// Mitsubishi GX Works2 project: EX_2_GROUP10   PLC: FX3G

// global labels: Global1
VAR_GLOBAL
  hopsInput AT D1120 : REAL;  (* input for hops inventory *)
  yeastQuantity AT D1130 : REAL;  (* yeast current quantity *)
  hopsQuantity AT D1150 : REAL;  (* hops current quantity *)
  startCooking AT X001 : BOOL;  (* starting stage 1 - cooking *)
  enoughIngredients AT M4 : BOOL;  (* if there is not quantity problem (enough required ingredients) *)
END_VAR
VAR_GLOBAL CONSTANT
  fermentationPilsnerTime : INT := 40;  (* fermentation time of Pilsner beer *)
  fermentationLagerTime : INT := 30;  (* fermentation time of Lager beer *)
  cookTime : INT := 40;  (* beer cook time last 4 seconds *)
  constant_0 : REAL;  (* constant zero *)
END_VAR
VAR_GLOBAL
  sampleValue AT D8201 : INT;  (* Sample value which symbolize the type of selected beer *)
END_VAR
VAR_GLOBAL CONSTANT
  normaliztionFactor : INT := 400;  (* normaliztion factor for the sampled value of beer kind *)
  maxLager : INT := 6;  (* Minimum sample value for lager beer (Underneath it is necessarily Pilsner beer) *)
  barleyLager : REAL := 12;  (* minimum quantity needed of barley for Lager beer *)
  hopsLager : REAL := 60;  (* minimum quantity needed of hops for Lager beer *)
  yeastPilsner : REAL := 120;  (* minimum quantity needed of yeast for Pilsner beer *)
  barleyPilsner : REAL := 6;  (* minimum quantity needed of barley for Pilsner beer *)
  hopsPilsner : REAL := 53;  (* minimum quantity needed of hops for Pilsner beer *)
END_VAR
VAR_GLOBAL
  barleyInput AT D1110 : REAL;  (* input for barley inventory *)
  yeastInput AT D1100 : REAL;  (* input for yeast inventory *)
  startDay AT X007 : BOOL;  (* start day button *)
  barleyQuantity AT D1140 : REAL;  (* barley current quantity *)
  yeast46Beers AT D1160 : REAL;  (* yeast demand for 6 beers *)
  barley46Beers AT D1170 : REAL;  (* barley demand for 6 beers *)
  cookContainer AT D2010 : REAL;  (* current quantity of raw materials in the cooking container *)
  emergencyButton AT X011 : BOOL;  (* emergency button that stopping the day (production process) *)
  workLed AT Y007 : BOOL;  (* led on until the day is finish *)
  fermentationTime AT D1190 : INT;  (* A variable indicating the required fermentation time *)
  hops46Beers AT D1180 : REAL;  (* hops demand for 6 beers *)
  analogInput_beerKind AT D8280 : INT;  (* analog input 1 value which determines which beer will produced *)
END_VAR
VAR_GLOBAL CONSTANT
  minBarley : REAL := 12;  (* minimum quantity needed of barley to produce beer *)
  minYeast : REAL := 150;  (* minimum quantity needed of yeast to produce beer *)
  minHops : REAL := 60;  (* minimum quantity needed of hops to produce beer *)
END_VAR
VAR_GLOBAL
  fermentationContainer AT D2020 : REAL;  (* current quantity of raw materials in fermentation container *)
END_VAR
VAR_GLOBAL CONSTANT
  yeastLager : REAL := 150;  (* minimum quantity needed of yeast for Lager beer *)
END_VAR
VAR_GLOBAL
  quantitiesProblem AT M1 : BOOL;  (* if NOT all input quantities are enough for starting the day or iteration *)
  keepTheDayOn AT M6 : BOOL;  (* auxiliary led - that X7 was pressed *)
  keepWork AT M7 : BOOL;  (* auxiliary led - there is no emargency *)
  finishSampleAnalog AT M10 : BOOL;  (* end of the sampling process for choosing the type of beer *)
  iterationDone AT M100 : BOOL;  (* full iteration tray production is done *)
  cookTimer4sec AT TC7 : BOOL;  (* counter 4 seconds for cooking time *)
  cookStop AT TS7 : BOOL;  (* cook timer is finished *)
  finishFillCookContainer AT M9 : BOOL;  (* finish transfer the raw materials from the stock to the cooking container *)
  pilsnerBeer AT M12 : BOOL;  (* beer kind is Pilsner *)
  lagerBeer AT M11 : BOOL;  (* beer kind is Lager *)
  stillCook AT Y001 : BOOL;  (* indicates that the cooking process is still in progress *)
  finishCooking AT M8 : BOOL;  (* stage 1 of cooking done *)
  InitBeerIngredients AT M13 : BOOL;  (* An auxiliary light for initializing the beer variables *)
  finishFillFerrnentationContainer AT M14 : BOOL;  (* finish transfer the raw materials from cooking container to the fermentation container *)
  timerReset1 AT M15 : BOOL;  (* reset timers after blinking *)
  endTimer1 AT TS5 : BOOL;  (* end timer for blinking Y3 *)
  timer1 AT TC5 : BOOL;  (* timer name for blinking time of Y3 *)
  fermentationLad1 AT Y003 : BOOL;  (* Indicator light for fermentation Lager beer *)
END_VAR
VAR_GLOBAL CONSTANT
  timeInterval : INT := 10;  (* time interval for light while blinking *)
END_VAR
VAR_GLOBAL
  counterSec AT TC8 : BOOL;  (* counter 4 or 3 seconds for fermentation time *)
  finishCounter AT TS8 : BOOL;  (* end timer for  fermentation time *)
  timer2 AT TC6 : BOOL;  (* timer name for blinking time of Y4 *)
  fermentationLad2 AT Y004 : BOOL;  (* Indicator light for fermentation Pilsner beer *)
  endTimer2 AT TS6 : BOOL;  (* end timer for blinking Y4 *)
  finishFermentation AT M16 : BOOL;  (* stage 2 of fermentation done *)
  startStorage AT X002 : BOOL;  (* starting stage 3 - Packing *)
  packCounter AT CC1 : BOOL;  (* counter for how many beers we pack in single iteration *)
END_VAR
VAR_GLOBAL CONSTANT
  packCounterValiueLast : INT := 6;  (* limit counter of 6 beers/ 1 package *)
END_VAR
VAR_GLOBAL
  packOneBeer AT X000 : BOOL;  (* Button for individual beer bottle packaging *)
  outCC1 AT CS1 : BOOL;  (* first press on X0 after starting packaging *)
  lastPackCounter AT CC2 : BOOL;  (* counter name of counter for last unit packing *)
  packingIsOn AT Y002 : BOOL;  (* Indication that packing a case of beers (six beers) is done *)
END_VAR
VAR_GLOBAL CONSTANT
  packCounterValiue : INT := 5;  (* counter indicating the packaging of all the case (six beers) *)
  packCounterValiueFirst : INT := 1;  (* counter indicating the packaging of the first beer in a case *)
END_VAR
VAR_GLOBAL
  outCC2 AT CS2 : BOOL;  (* finish 6 press on X0 after starting packaging *)
END_VAR
VAR_GLOBAL CONSTANT
  OnePackageReady : INT := 1;  (* constant- insert one package to packages of beer *)
END_VAR
VAR_GLOBAL
  readyBeerPack AT D2040 : INT;  (* number of prepared packages of beer *)
  fermentationStart AT X005 : BOOL;  (* starting stage 2 -fermentation *)
END_VAR
VAR_GLOBAL CONSTANT
  normaliztionFactor2 : INT := 40;  (* normaliztion factor for the number of beers produced (decimal representation) *)
END_VAR
VAR_GLOBAL
  beerPackOutput AT D8282 : INT;  (* output for the number o ready beers packages in tens *)
END_VAR
VAR_GLOBAL CONSTANT
  constantWord_0 : INT;  (* constant zero kind word *)
END_VAR

// task Task_01 (event TRUE, interval 0, priority 31): POU_01

PROGRAM POU_01
(* structured ladder/FBD written out as ST: instructions are called as NAME(EN, inputs, outputs); _pN, _eN, _tN stand for wires *)
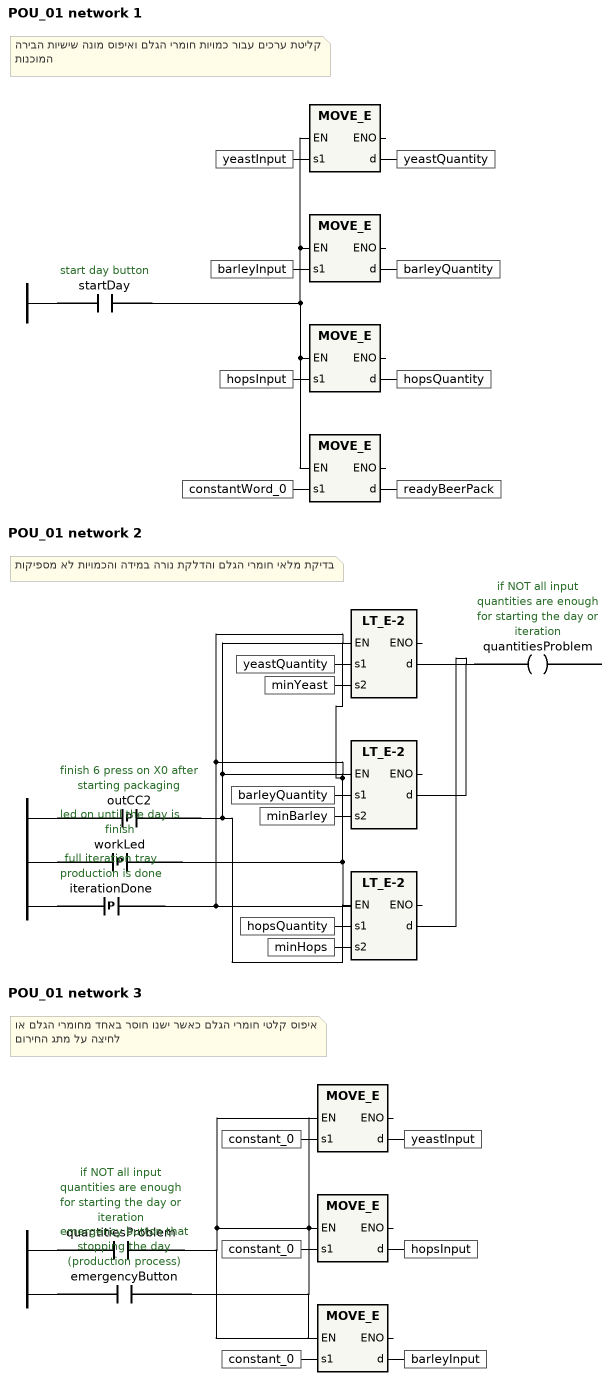
(* network 1 *)
(* קליטת ערכים עבור כמויות חומרי הגלם ואיפוס מונה שישיות הבירה המוכנות *)
MOVE_E(startDay, yeastInput, yeastQuantity);
MOVE_E(startDay, barleyInput, barleyQuantity);
MOVE_E(startDay, hopsInput, hopsQuantity);
MOVE_E(startDay, constantWord_0, readyBeerPack);
(* network 2 *)
(* בדיקת מלאי חומרי הגלם והדלקת נורה במידה והכמויות לא מספיקות *)
_p1 := LDP(TRUE, outCC2) OR LDP(TRUE, workLed) OR LDP(TRUE, iterationDone);
LT_E(_p1, yeastQuantity, minYeast, _t2);
LT_E(_p1, barleyQuantity, minBarley, _t3);
LT_E(_p1, hopsQuantity, minHops, _t4);
quantitiesProblem := _t2 OR _t3 OR _t4;
(* network 3 *)
(* איפוס קלטי חומרי הגלם כאשר ישנו חוסר באחד מחומרי הגלם או לחיצה על מתג החירום *)
_p1 := quantitiesProblem OR emergencyButton;
MOVE_E(_p1, constant_0, yeastInput);
MOVE_E(_p1, constant_0, hopsInput);
MOVE_E(_p1, constant_0, barleyInput);
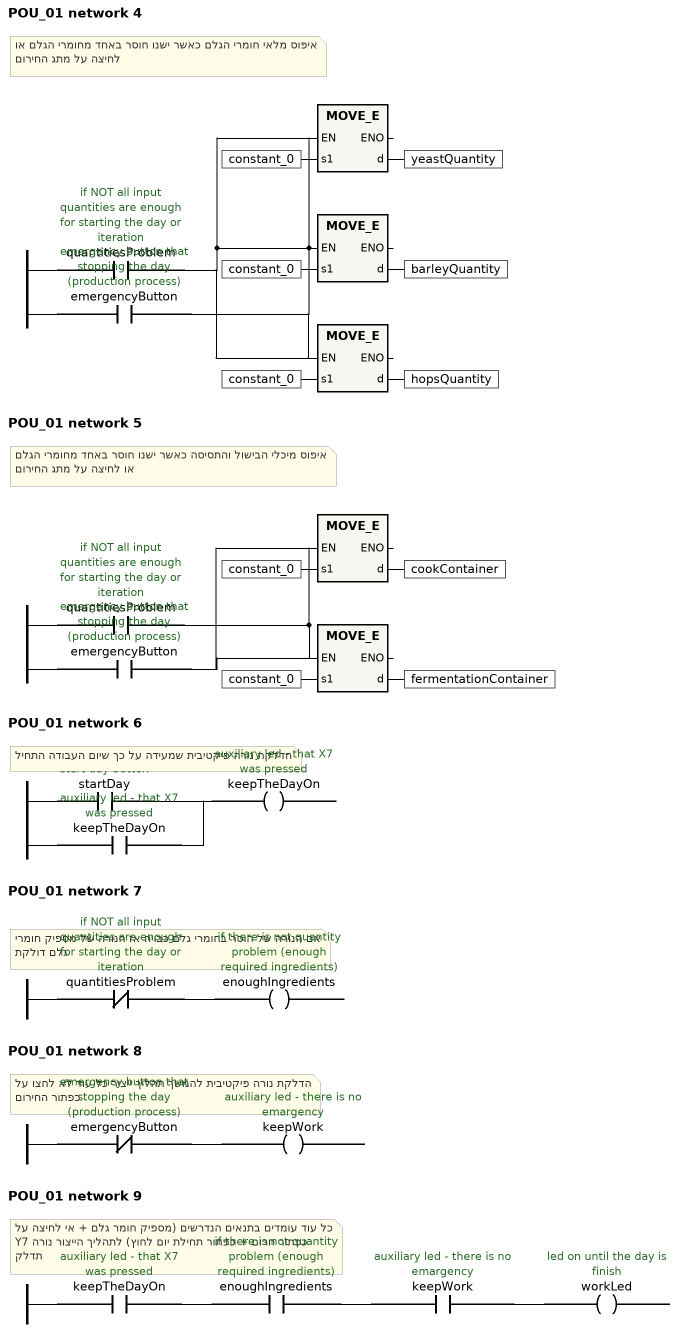
(* network 4 *)
(* איפוס מלאי חומרי הגלם כאשר ישנו חוסר באחד מחומרי הגלם או לחיצה על מתג החירום *)
_p1 := quantitiesProblem OR emergencyButton;
MOVE_E(_p1, constant_0, yeastQuantity);
MOVE_E(_p1, constant_0, barleyQuantity);
MOVE_E(_p1, constant_0, hopsQuantity);
(* network 5 *)
(* איפוס מיכלי הבישול והתסיסה כאשר ישנו חוסר באחד מחומרי הגלם או לחיצה על מתג החירום *)
_p1 := quantitiesProblem OR emergencyButton;
MOVE_E(_p1, constant_0, cookContainer);
MOVE_E(_p1, constant_0, fermentationContainer);
(* network 6 *)
(* הדלקת נורה פיקטיבית שמעידה על כך שיום העבודה התחיל *)
keepTheDayOn := startDay OR keepTheDayOn;
(* network 7 *)
(* אם הנורה של חוסר בחומרי גלם כבויה אז הנורה של מספיק חומרי גלם דולקת *)
enoughIngredients := NOT quantitiesProblem;
(* network 8 *)
(* הדלקת נורה פיקטיבית להמשך תהליך ייצור כל עוד לא לחצו על כפתור החירום *)
keepWork := NOT emergencyButton;
(* network 9 *)
(* כל עוד עומדים בתנאים הנדרשים (מספיק חומר גלם + אי לחיצה על כפתור חרום + כפתור תחילת יום לחוץ) לתהליך הייצור נורה Y7 תדלק *)
workLed := keepTheDayOn AND enoughIngredients AND keepWork;
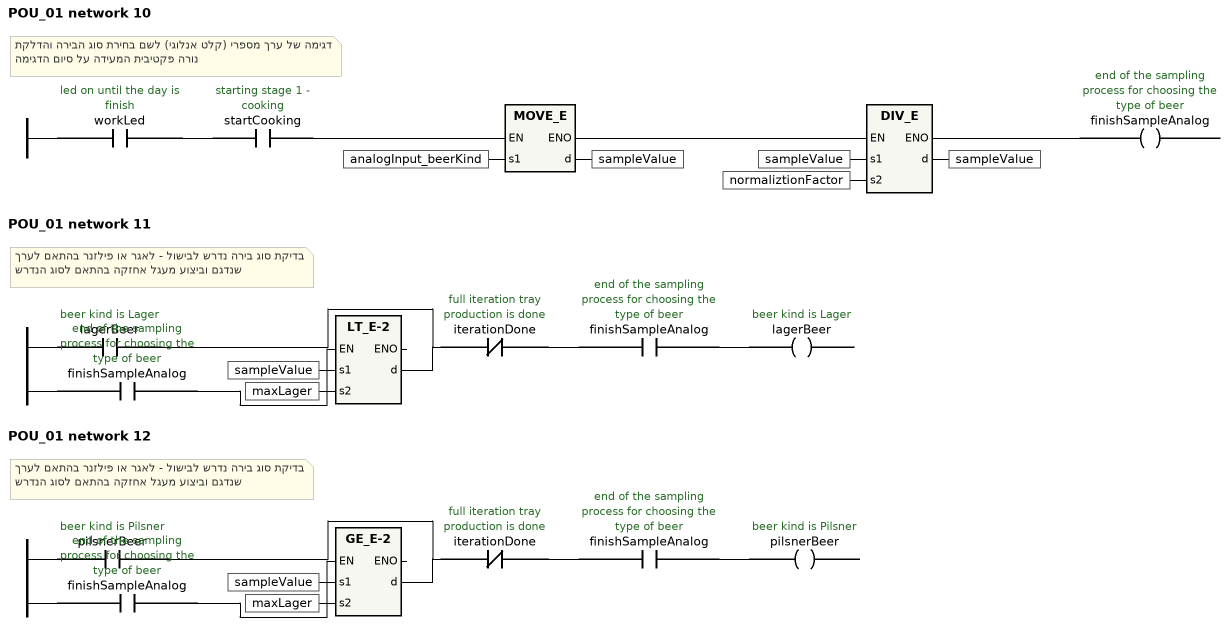
(* network 10 *)
(* דגימה של ערך מספרי (קלט אנלוגי) לשם בחירת סוג הבירה והדלקת נורה פקטיבית המעידה על סיום הדגימה *)
_e1 := MOVE_E(workLed AND startCooking, analogInput_beerKind, sampleValue);
_e2 := DIV_E(_e1, sampleValue, normaliztionFactor, sampleValue);
finishSampleAnalog := _e2;
(* network 11 *)
(* בדיקת סוג בירה נדרש לבישול - לאגר או פילזנר בהתאם לערך שנדגם וביצוע מעגל אחזקה בהתאם לסוג הנדרש *)
LT_E(finishSampleAnalog, sampleValue, maxLager, _t1);
lagerBeer := ((lagerBeer OR _t1) AND NOT iterationDone) AND finishSampleAnalog;
(* network 12 *)
(* בדיקת סוג בירה נדרש לבישול - לאגר או פילזנר בהתאם לערך שנדגם וביצוע מעגל אחזקה בהתאם לסוג הנדרש *)
GE_E(finishSampleAnalog, sampleValue, maxLager, _t1);
pilsnerBeer := ((pilsnerBeer OR _t1) AND NOT iterationDone) AND finishSampleAnalog;
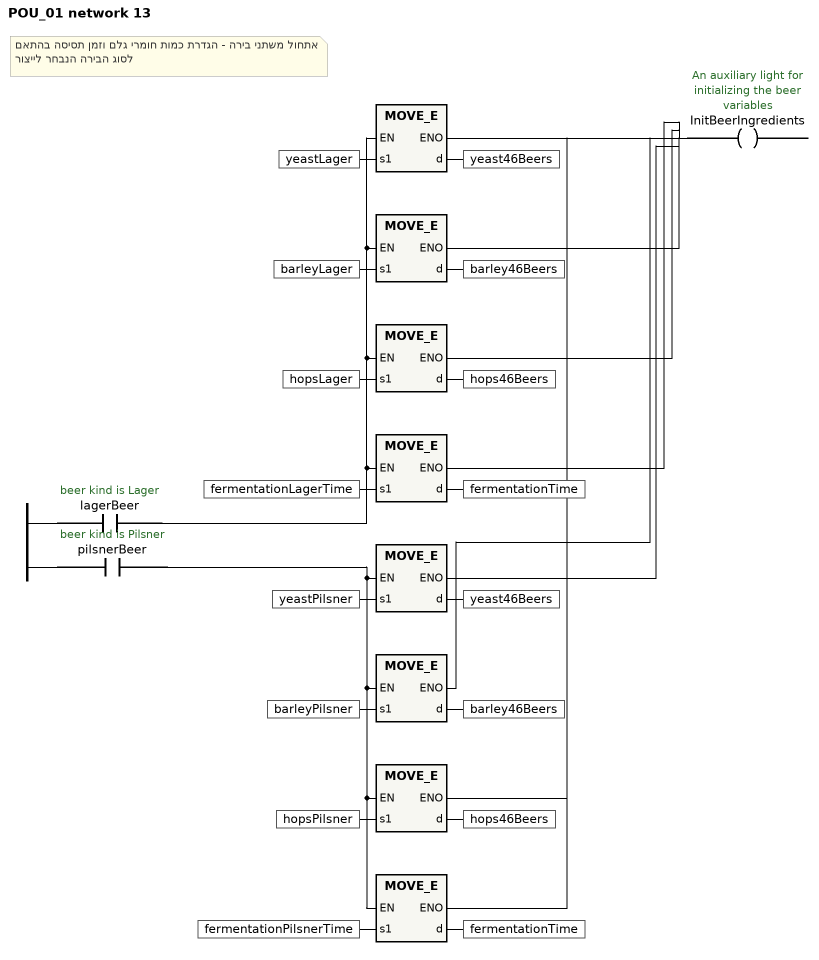
(* network 13 *)
(* אתחול משתני בירה - הגדרת כמות חומרי גלם וזמן תסיסה בהתאם לסוג הבירה הנבחר לייצור *)
_e1 := MOVE_E(lagerBeer, yeastLager, yeast46Beers);
_e2 := MOVE_E(lagerBeer, barleyLager, barley46Beers);
_e3 := MOVE_E(lagerBeer, hopsLager, hops46Beers);
_e4 := MOVE_E(lagerBeer, fermentationLagerTime, fermentationTime);
_e5 := MOVE_E(pilsnerBeer, yeastPilsner, yeast46Beers);
_e6 := MOVE_E(pilsnerBeer, barleyPilsner, barley46Beers);
_e7 := MOVE_E(pilsnerBeer, hopsPilsner, hops46Beers);
_e8 := MOVE_E(pilsnerBeer, fermentationPilsnerTime, fermentationTime);
InitBeerIngredients := _e1 OR _e2 OR _e3 OR _e4 OR _e5 OR _e6 OR _e7 OR _e8;
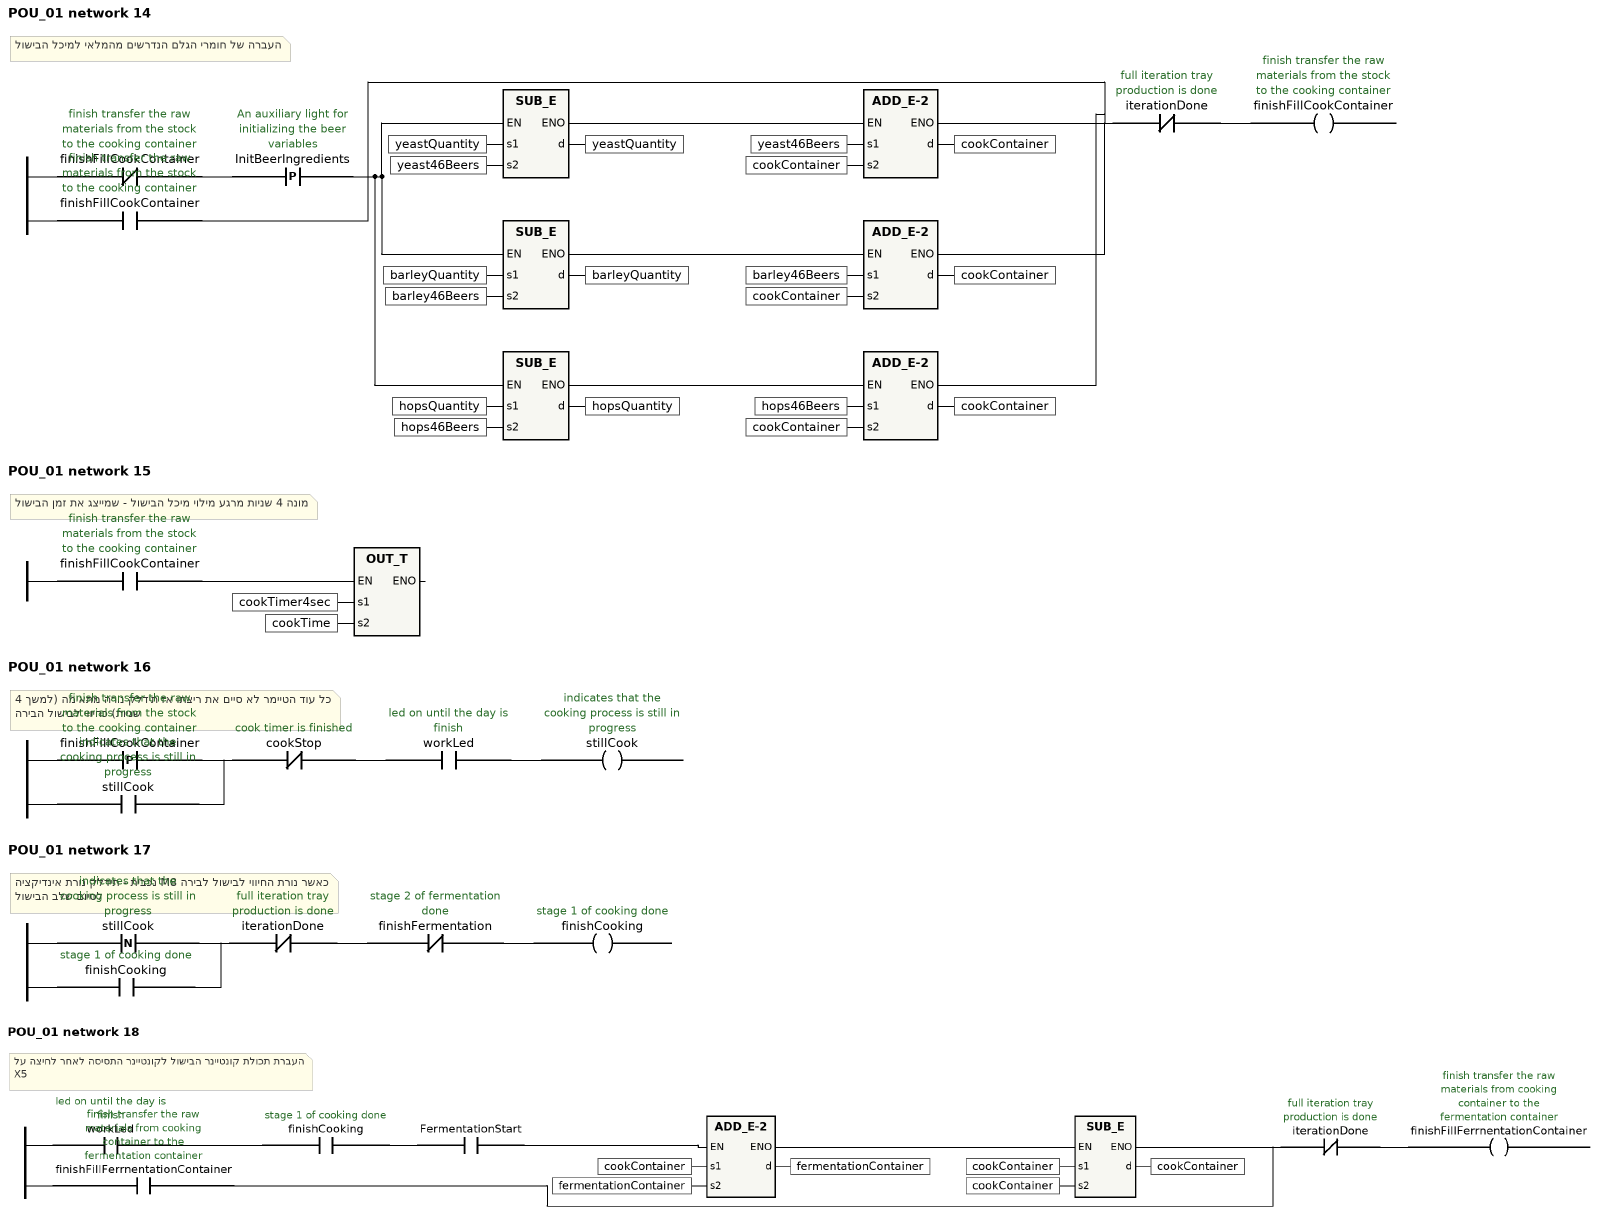
(* network 14 *)
(* העברה של חומרי הגלם הנדרשים מהמלאי למיכל הבישול *)
_p1 := NOT finishFillCookContainer AND LDP(TRUE, InitBeerIngredients);
_e2 := SUB_E(_p1, yeastQuantity, yeast46Beers, yeastQuantity);
_e3 := ADD_E(_e2, yeast46Beers, cookContainer, cookContainer);
_e4 := SUB_E(_p1, barleyQuantity, barley46Beers, barleyQuantity);
_e5 := ADD_E(_e4, barley46Beers, cookContainer, cookContainer);
_e6 := SUB_E(_p1, hopsQuantity, hops46Beers, hopsQuantity);
_e7 := ADD_E(_e6, hops46Beers, cookContainer, cookContainer);
finishFillCookContainer := (_e3 OR _e5 OR _e7 OR finishFillCookContainer) AND NOT iterationDone;
(* network 15 *)
(* מונה 4 שניות מרגע מילוי מיכל הבישול - שמייצג את זמן הבישול *)
OUT_T(finishFillCookContainer, cookTimer4sec, cookTime);
(* network 16 *)
(* כל עוד הטיימר לא סיים את ריצתו אז תידלק נורה מתאימה (למשך 4 שניות) כחיווי לבישול הבירה *)
stillCook := ((LDP(TRUE, finishFillCookContainer) OR stillCook) AND NOT cookStop) AND workLed;
(* network 17 *)
(* כאשר נורת החיווי לבישול לבירה M8 נכבית - תידלק נורת אינדיקציה לסיום שלב הבישול *)
finishCooking := ((LDF(TRUE, stillCook) OR finishCooking) AND NOT iterationDone) AND NOT finishFermentation;
(* network 18 *)
(* העברת תכולת קונטיינר הבישול לקונטיינר התסיסה לאחר לחיצה על X5 *)
_e1 := ADD_E(workLed AND finishCooking AND FermentationStart, cookContainer, fermentationContainer, fermentationContainer);
_e2 := SUB_E(_e1, cookContainer, cookContainer, cookContainer);
finishFillFerrnentationContainer := (_e2 OR finishFillFerrnentationContainer) AND NOT iterationDone;
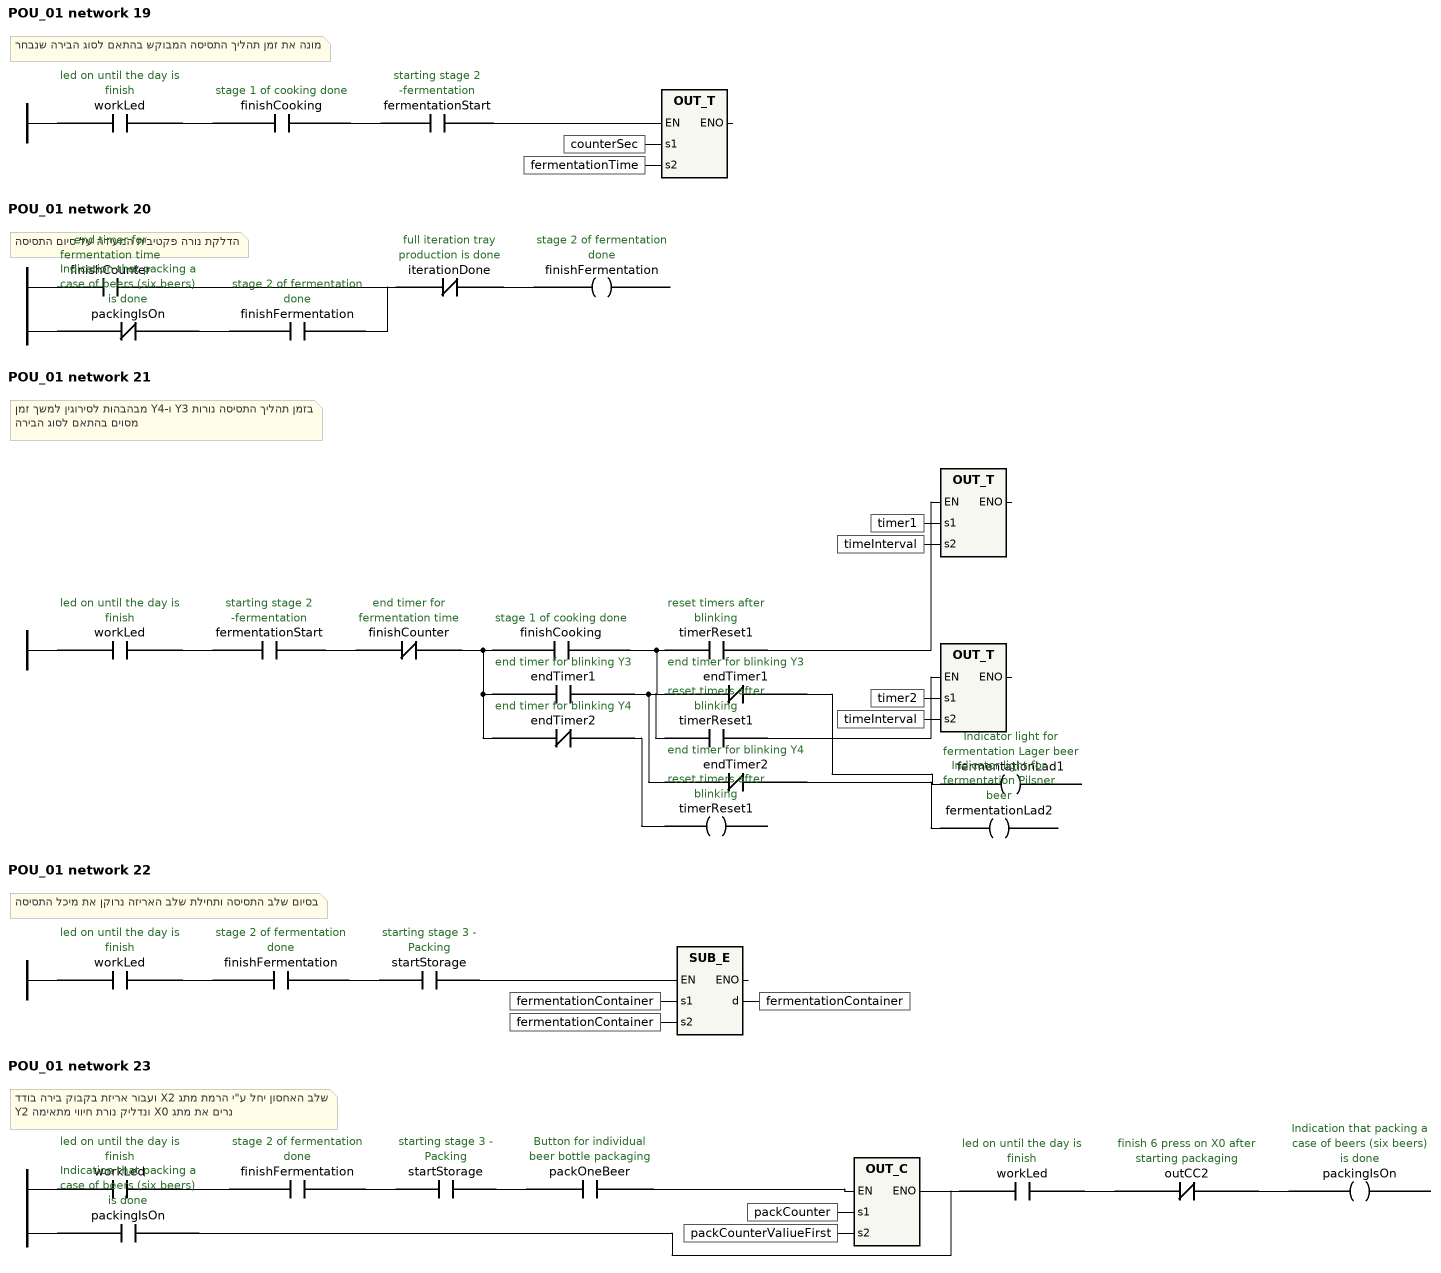
(* network 19 *)
(* מונה את זמן תהליך התסיסה המבוקש בהתאם לסוג הבירה שנבחר *)
OUT_T(workLed AND finishCooking AND fermentationStart, counterSec, fermentationTime);
(* network 20 *)
(* הדלקת נורה פקטיבית המעידה על סיום התסיסה *)
finishFermentation := (finishCounter OR (NOT packingIsOn AND finishFermentation)) AND NOT iterationDone;
(* network 21 *)
(* בזמן תהליך התסיסה נורות Y3 ו-Y4 מבהבהות לסירוגין למשך זמן מסוים בהתאם לסוג הבירה *)
_p1 := workLed AND fermentationStart AND NOT finishCounter;
_p2 := _p1 AND finishCooking;
OUT_T(_p2 AND timerReset1, timer1, timeInterval);
fermentationLad1 := _p2 AND NOT endTimer1;
_p3 := _p1 AND endTimer1;
OUT_T(_p3 AND timerReset1, timer2, timeInterval);
fermentationLad2 := _p3 AND NOT endTimer2;
timerReset1 := _p1 AND NOT endTimer2;
(* network 22 *)
(* בסיום שלב התסיסה ותחילת שלב האריזה נרוקן את מיכל התסיסה *)
SUB_E(workLed AND finishFermentation AND startStorage, fermentationContainer, fermentationContainer, fermentationContainer);
(* network 23 *)
(* שלב האחסון יחל ע"י הרמת מתג X2 ועבור אריזת בקבוק בירה בודד נרים את מתג X0 ונדליק נורת חיווי מתאימה Y2 *)
_e1 := OUT_C(workLed AND finishFermentation AND startStorage AND packOneBeer, packCounter, packCounterValiueFirst);
packingIsOn := ((_e1 OR packingIsOn) AND workLed) AND NOT outCC2;
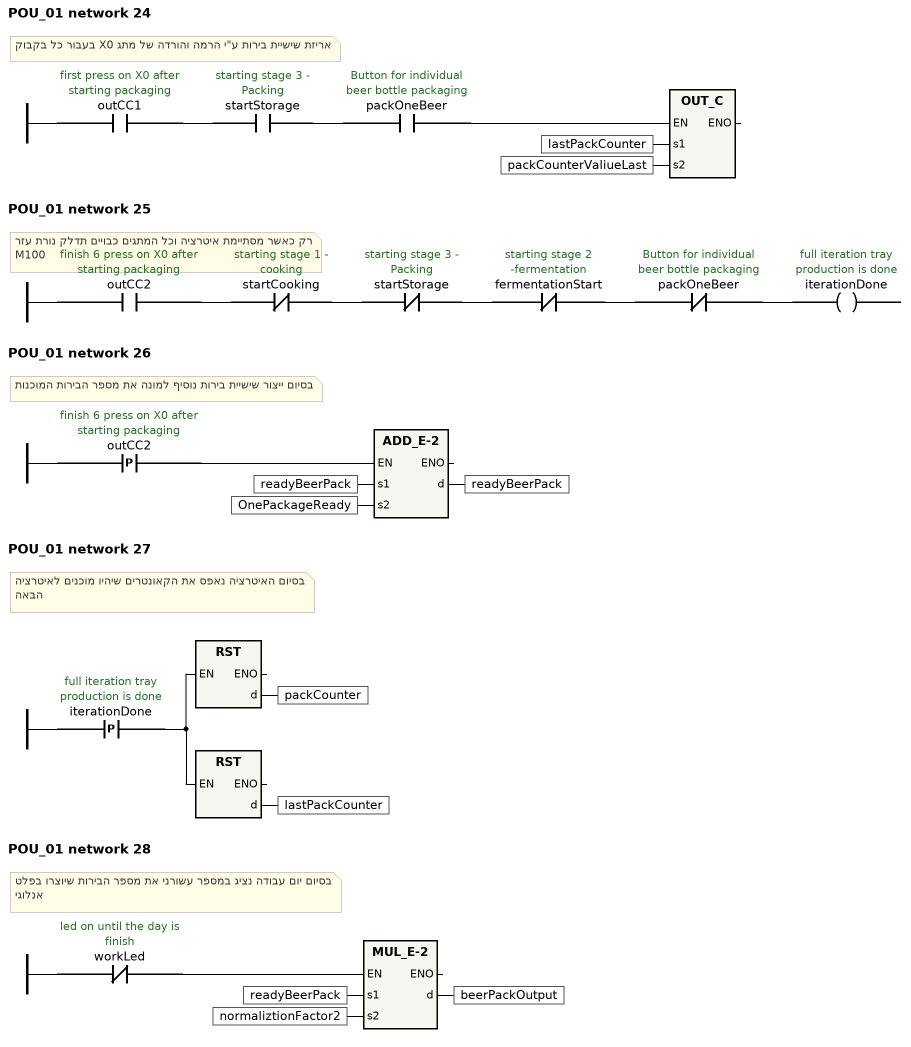
(* network 24 *)
(* אריזת שישיית בירות ע"י הרמה והורדה של מתג X0 בעבור כל בקבוק *)
OUT_C(outCC1 AND startStorage AND packOneBeer, lastPackCounter, packCounterValiueLast);
(* network 25 *)
(* רק כאשר מסתיימת איטרציה וכל המתגים כבויים תדלק נורת עזר M100 *)
iterationDone := outCC2 AND NOT startCooking AND NOT startStorage AND NOT fermentationStart AND NOT packOneBeer;
(* network 26 *)
(* בסיום ייצור שישיית בירות נוסיף למונה את מספר הבירות המוכנות *)
ADD_E(LDP(TRUE, outCC2), readyBeerPack, OnePackageReady, readyBeerPack);
(* network 27 *)
(* בסיום האיטרציה נאפס את הקאונטרים שיהיו מוכנים לאיטרציה הבאה *)
_p1 := LDP(TRUE, iterationDone);
RST(_p1, packCounter);
RST(_p1, lastPackCounter);
(* network 28 *)
(* בסיום יום עבודה נציג במספר עשורני את מספר הבירות שיוצרו בפלט אנלוגי *)
MUL_E(NOT workLed, readyBeerPack, normaliztionFactor2, beerPackOutput);
END_PROGRAM
